// TIA Portal project "64396156_S7-1200_DataLogging_PROJ_v2d0" (V14)

(* hardware
DEVICE "SIMATIC 1200-Station_1"  S71200.Device
   slot 0: "S7-1200 rack"  Rack  V1.0
   slot 1: "PLC_1"  CPU 1211C DC/DC/DC  6ES7 211-1AE40-0XB0  V4.2
*)

// ===== PLC "PLC_1"  CPU 1211C DC/DC/DC =====

VAR_GLOBAL   // PLC tag table "Standard-Variablentabelle"
   "System_Byte" AT %MB1 : Byte;
   "FirstScan" AT %M1.0 : Bool;
   "DiagStatusUpdate" AT %M1.1 : Bool;
   "AlwaysTRUE" AT %M1.2 : Bool;
   "AlwaysFALSE" AT %M1.3 : Bool;
   "Clock_Byte" AT %MB0 : Byte;
   "Clock_10Hz" AT %M0.0 : Bool;
   "Clock_5Hz" AT %M0.1 : Bool;
   "Clock_2.5Hz" AT %M0.2 : Bool;
   "Clock_2Hz" AT %M0.3 : Bool;
   "Clock_1.25Hz" AT %M0.4 : Bool;
   "Clock_1Hz" AT %M0.5 : Bool;
   "Clock_0.625Hz" AT %M0.6 : Bool;
   "Clock_0.5Hz" AT %M0.7 : Bool;
END_VAR

TYPE "BLOCK"
VERSION : 0.1
   STRUCT
      REQ : Bool;
      DONE : Bool;
      BUSY : Bool;
      ERROR : Bool;
      STATUS : Word;
   END_STRUCT;
END_TYPE

TYPE "Type_SndParam"
VERSION : 0.1
   STRUCT
      interfaceId : Hw_Any;   // Hardware identifier
      conId : Conn_Ouc;   // Connection ID
      phoneNumber : String[22];   // Phone number
      smsText : String[160];   // Sms Text
   END_STRUCT;
END_TYPE

DATA_BLOCK "Tags"   // DB147
{ S7_Optimized_Access := 'TRUE' }
VERSION : 0.1
   VAR
      T : Struct
         Temperature : Real;
         Offset : Real := -22.0;
         Amplitude : Real := 6.0;
         Period : Real := 600.0;
      END_STRUCT;
   END_VAR
   VAR RETAIN
      DataLog : Struct
         Enable : Bool := true;
         Reset : Bool;
         DATA : Struct
            Temperature : Real;
         END_STRUCT;
         State : USInt;
         ErrorStatus : Word;
         NumberRecords : UDInt;
         CurrentName : String;
         WriteDone : Bool;
      END_STRUCT;
      TmailC : Struct
         Enable : Bool := false;
         Temperature_max : Real := -20.0;
         Reset : Bool;
         State : USInt;
         ErrorStatus : Word;
         ErrorCounter : UDInt;
         DoneCounter : UDInt;
      END_STRUCT;
   END_VAR
   VAR
      sms : Struct
         enable : Bool;
         sndSmsParam : "Type_SndParam";
         sndSmsOB1 : Bool;   // Bit, which activates Snd Sms block
         doneSndOB1 : Bool;   // Done. Signal for one progrmm cycle active
         busySndOB1 : Bool;   // Block is active
         errorSndOB1 : Bool;   // Error. Signal for one cycle active
         statusSndOB1 : DWord;   // Error Status for one Program cycle active
      END_STRUCT;
   END_VAR
BEGIN
   sms.sndSmsParam.smsText := 'The temperature is too high! Please check the system.';
   sms.sndSmsParam.phoneNumber := '+4915150006535';
   sms.sndSmsParam.conId := 1;
   sms.sndSmsParam.interfaceId := 270;
END_DATA_BLOCK

// folder: DataLog

DATA_BLOCK "DataLog_DB"   // DB143
{ S7_Optimized_Access := 'TRUE' }
VERSION : 0.1
// stored: InstanceOfName DataLog
"DataLog"
BEGIN
END_DATA_BLOCK

// folder: Simulation

DATA_BLOCK "T_simulation_DB"   // DB148
{ S7_Optimized_Access := 'TRUE' }
VERSION : 0.1
// stored: InstanceOfName T_simulation
"T_simulation"
BEGIN
END_DATA_BLOCK

// folder: TmailC

DATA_BLOCK "TmailC_DB"   // DB149
{ S7_Optimized_Access := 'TRUE' }
VERSION : 0.1
// stored: InstanceOfName TmailC
"TmailC"
BEGIN
END_DATA_BLOCK

// folder: (top level)

ORGANIZATION_BLOCK "Main"   // OB1, FBD, ProgramCycle
TITLE = "Main Program Sweep (Cycle)"
{ S7_Optimized_Access := 'TRUE' }
VERSION : 0.1
   VAR_INPUT
      Initial_Call : Bool;   // Initial call of this OB
      Remanence : Bool;   // =True, if remanent data are available
   END_VAR
BEGIN

REGION Network 1: Temperature simulation
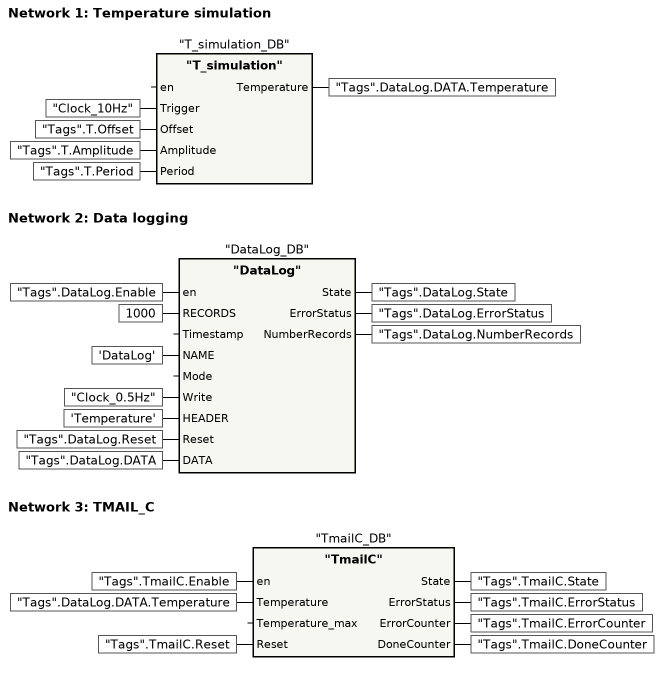
   "T_simulation_DB"(Trigger := "Clock_10Hz",   // "T_simulation"
                     Offset := "Tags".T.Offset,
                     Amplitude := "Tags".T.Amplitude,
                     Period := "Tags".T.Period,
                     Temperature => "Tags".DataLog.DATA.Temperature);
END_REGION

REGION Network 2: Data logging
   IF "Tags".DataLog.Enable THEN
       "DataLog_DB"(RECORDS := 1000,   // "DataLog"
                    "NAME" := 'DataLog',
                    Write := "Clock_0.5Hz",
                    HEADER := 'Temperature',
                    Reset := "Tags".DataLog.Reset,
                    DATA := "Tags".DataLog.DATA,
                    State => "Tags".DataLog.State,
                    ErrorStatus => "Tags".DataLog.ErrorStatus,
                    NumberRecords => "Tags".DataLog.NumberRecords);
   END_IF;
END_REGION

REGION Network 3: TMAIL_C
   IF "Tags".TmailC.Enable THEN
       "TmailC_DB"(Temperature := "Tags".DataLog.DATA.Temperature,   // "TmailC"
                   Reset := "Tags".TmailC.Reset,
                   State => "Tags".TmailC.State,
                   ErrorStatus => "Tags".TmailC.ErrorStatus,
                   ErrorCounter => "Tags".TmailC.ErrorCounter,
                   DoneCounter => "Tags".TmailC.DoneCounter);
   END_IF;
END_REGION
END_ORGANIZATION_BLOCK

// folder: DataLog

FUNCTION_BLOCK "DataLog"   // FB143, LAD
{ S7_Optimized_Access := 'TRUE' }
VERSION : 0.1
   VAR_INPUT
      RECORDS : UDInt;
      Timestamp : Bool := true;
      "NAME" : String;
      Mode : Bool;
      Write : Bool;
      HEADER : String;
      Reset : Bool;
   END_VAR
   VAR_OUTPUT
      State : USInt;
      ErrorStatus : Word;
      NumberRecords : UDInt;
   END_VAR
   VAR_IN_OUT
      DATA : Variant;
   END_VAR
   VAR RETAIN
      ID : UDInt;
      "Step" : USInt;
   END_VAR
   VAR
      CreateB : "BLOCK";
      OpenB : "BLOCK";
      WriteB : "BLOCK";
      write_edge : Bool;
   END_VAR
   VAR RETAIN
      NumberRecords_inout : UDInt;
   END_VAR
   VAR
      HEADER_inout : String;
      DataLogCreate_Instance : DataLogCreate;
      DataLogOpen_Instance : DataLogOpen;
      DataLogWrite_Instance : DataLogWrite;
      tmp_TIMESTAMP : UInt;
      tmp_MODE : UInt;
   END_VAR
   VAR_TEMP   // added for the SCL form of the ladder/FBD networks
      _w1 : Bool;
      _w2 : Bool;
      _w3 : Bool;
   END_VAR
BEGIN

REGION Network 1: Command 0: Create
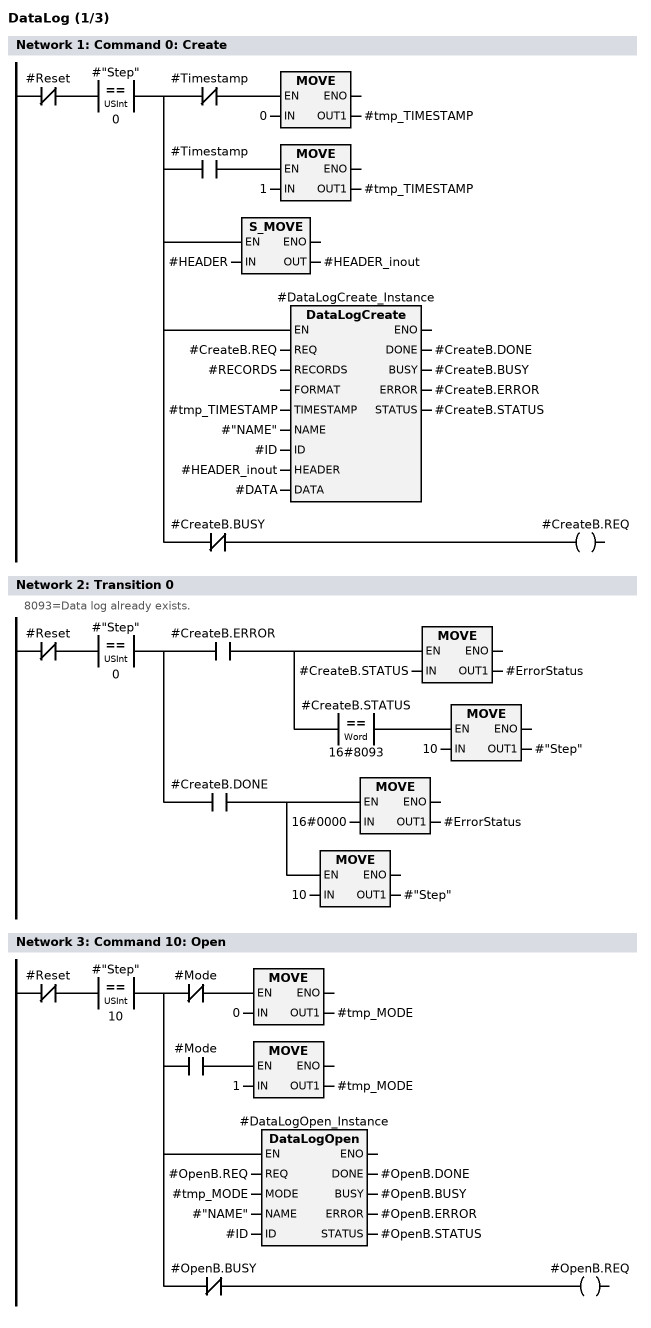
   #_w1 := NOT #Reset AND (#"Step" = 0);
   IF #_w1 AND NOT #Timestamp THEN #tmp_TIMESTAMP := 0; END_IF;
   IF #_w1 AND #Timestamp THEN #tmp_TIMESTAMP := 1; END_IF;
   IF #_w1 THEN
       #HEADER_inout := #HEADER;
       #DataLogCreate_Instance(REQ := #CreateB.REQ,   // DataLogCreate
                               RECORDS := #RECORDS,
                               TIMESTAMP := #tmp_TIMESTAMP,
                               "NAME" := #"NAME",
                               ID := #ID,
                               HEADER := #HEADER_inout,
                               DATA := #DATA,
                               DONE => #CreateB.DONE,
                               BUSY => #CreateB.BUSY,
                               ERROR => #CreateB.ERROR,
                               STATUS => #CreateB.STATUS);
   END_IF;
   #CreateB.REQ := #_w1 AND NOT #CreateB.BUSY;
END_REGION

REGION Network 2: Transition 0
   // 8093=Data log already exists.
   RUNG wire#powerrail
      I_Contact( #Reset )
      { S7_Templates := "SrcType := USInt" } EQ_Contact(in1 := #"Step", in2 := 0)
      wire#w1
      Contact( #CreateB.ERROR )
      wire#w2
      { S7_GenerateENO := "TRUE" } Move(in := #CreateB.STATUS, out1 => #ErrorStatus)
   END_RUNG
   RUNG wire#w2
      { S7_Templates := "SrcType := Word" } EQ_Contact(in1 := #CreateB.STATUS, in2 := 16#8093)
      { S7_GenerateENO := "TRUE" } Move(in := 10, out1 => #"Step")
   END_RUNG
   RUNG wire#w1
      Contact( #CreateB.DONE )
      wire#w3
      { S7_GenerateENO := "TRUE" } Move(in := 16#0000, out1 => #ErrorStatus)
   END_RUNG
   RUNG wire#w3
      { S7_GenerateENO := "TRUE" } Move(in := 10, out1 => #"Step")
   END_RUNG
   // the same network as SCL:
   #_w1 := NOT #Reset AND (#"Step" = 0);
   #_w2 := #_w1 AND #CreateB.ERROR;
   IF #_w2 THEN #ErrorStatus := #CreateB.STATUS; END_IF;
   IF #_w2 AND (#CreateB.STATUS = 16#8093) THEN #"Step" := 10; END_IF;
   IF #_w1 AND #CreateB.DONE THEN
       #ErrorStatus := 16#0000;
       #"Step" := 10;
   END_IF;
END_REGION

REGION Network 3: Command 10: Open
   #_w1 := NOT #Reset AND (#"Step" = 10);
   IF #_w1 AND NOT #Mode THEN #tmp_MODE := 0; END_IF;
   IF #_w1 AND #Mode THEN #tmp_MODE := 1; END_IF;
   IF #_w1 THEN
       #DataLogOpen_Instance(REQ := #OpenB.REQ,   // DataLogOpen
                             MODE := #tmp_MODE,
                             "NAME" := #"NAME",
                             ID := #ID,
                             DONE => #OpenB.DONE,
                             BUSY => #OpenB.BUSY,
                             ERROR => #OpenB.ERROR,
                             STATUS => #OpenB.STATUS);
   END_IF;
   #OpenB.REQ := #_w1 AND NOT #OpenB.BUSY;
END_REGION

REGION Network 4: Transition 10
   // 8092=Data log does not exist
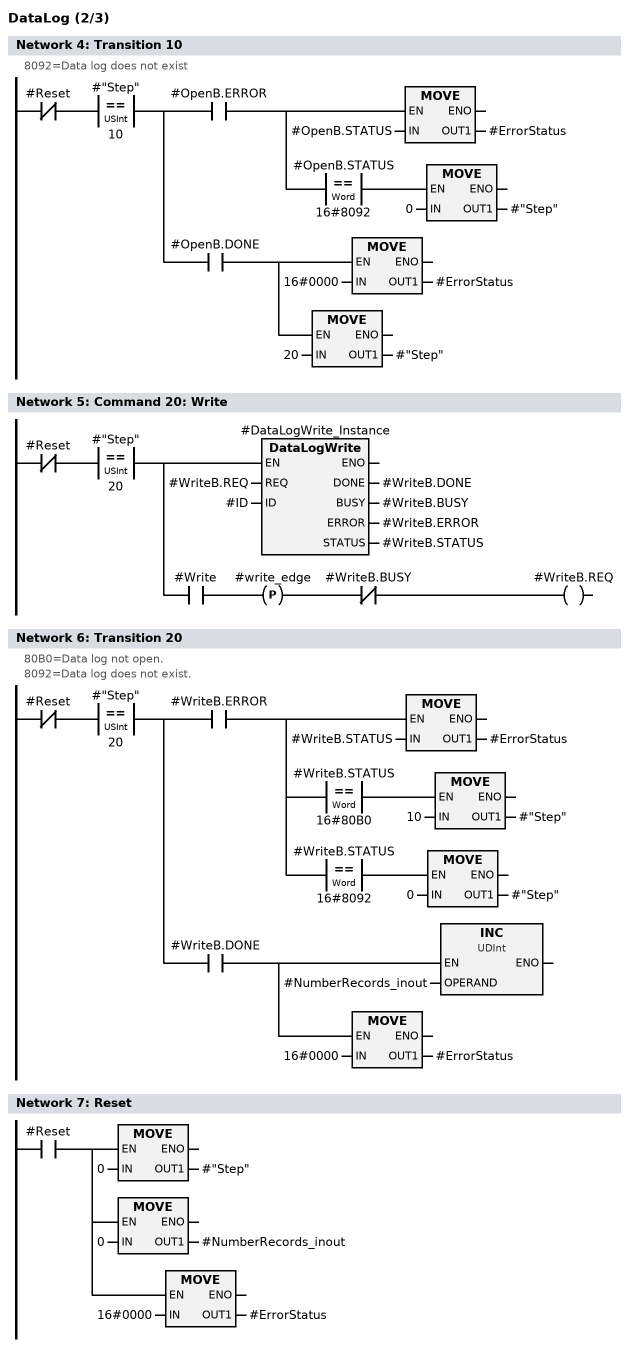
   RUNG wire#powerrail
      I_Contact( #Reset )
      { S7_Templates := "SrcType := USInt" } EQ_Contact(in1 := #"Step", in2 := 10)
      wire#w1
      Contact( #OpenB.ERROR )
      wire#w2
      { S7_GenerateENO := "TRUE" } Move(in := #OpenB.STATUS, out1 => #ErrorStatus)
   END_RUNG
   RUNG wire#w2
      { S7_Templates := "SrcType := Word" } EQ_Contact(in1 := #OpenB.STATUS, in2 := 16#8092)
      { S7_GenerateENO := "TRUE" } Move(in := 0, out1 => #"Step")
   END_RUNG
   RUNG wire#w1
      Contact( #OpenB.DONE )
      wire#w3
      { S7_GenerateENO := "TRUE" } Move(in := 16#0000, out1 => #ErrorStatus)
   END_RUNG
   RUNG wire#w3
      { S7_GenerateENO := "TRUE" } Move(in := 20, out1 => #"Step")
   END_RUNG
   // the same network as SCL:
   #_w1 := NOT #Reset AND (#"Step" = 10);
   #_w2 := #_w1 AND #OpenB.ERROR;
   IF #_w2 THEN #ErrorStatus := #OpenB.STATUS; END_IF;
   IF #_w2 AND (#OpenB.STATUS = 16#8092) THEN #"Step" := 0; END_IF;
   IF #_w1 AND #OpenB.DONE THEN
       #ErrorStatus := 16#0000;
       #"Step" := 20;
   END_IF;
END_REGION

REGION Network 5: Command 20: Write
   #_w1 := NOT #Reset AND (#"Step" = 20);
   IF #_w1 THEN
       #DataLogWrite_Instance(REQ := #WriteB.REQ,   // DataLogWrite
                              ID := #ID,
                              DONE => #WriteB.DONE,
                              BUSY => #WriteB.BUSY,
                              ERROR => #WriteB.ERROR,
                              STATUS => #WriteB.STATUS);
   END_IF;
   #_w2 := #_w1 AND #Write;
   #_w3 := #_w2 AND NOT #write_edge;   // rising edge
   #write_edge := #_w2;
   #WriteB.REQ := #_w3 AND NOT #WriteB.BUSY;
END_REGION

REGION Network 6: Transition 20
   // 80B0=Data log not open.
   // 8092=Data log does not exist.
   RUNG wire#powerrail
      I_Contact( #Reset )
      { S7_Templates := "SrcType := USInt" } EQ_Contact(in1 := #"Step", in2 := 20)
      wire#w1
      Contact( #WriteB.ERROR )
      wire#w2
      { S7_GenerateENO := "TRUE" } Move(in := #WriteB.STATUS, out1 => #ErrorStatus)
   END_RUNG
   RUNG wire#w2
      { S7_Templates := "SrcType := Word" } EQ_Contact(in1 := #WriteB.STATUS, in2 := 16#80B0)
      { S7_GenerateENO := "TRUE" } Move(in := 10, out1 => #"Step")
   END_RUNG
   RUNG wire#w2
      { S7_Templates := "SrcType := Word" } EQ_Contact(in1 := #WriteB.STATUS, in2 := 16#8092)
      { S7_GenerateENO := "TRUE" } Move(in := 0, out1 => #"Step")
   END_RUNG
   RUNG wire#w1
      Contact( #WriteB.DONE )
      wire#w3
      { S7_Templates := "DestType := UDInt"; S7_GenerateENO := "TRUE" } Inc( #NumberRecords_inout )
   END_RUNG
   RUNG wire#w3
      { S7_GenerateENO := "TRUE" } Move(in := 16#0000, out1 => #ErrorStatus)
   END_RUNG
   // the same network as SCL:
   #_w1 := NOT #Reset AND (#"Step" = 20);
   #_w2 := #_w1 AND #WriteB.ERROR;
   IF #_w2 THEN #ErrorStatus := #WriteB.STATUS; END_IF;
   IF #_w2 AND (#WriteB.STATUS = 16#80B0) THEN #"Step" := 10; END_IF;
   IF #_w2 AND (#WriteB.STATUS = 16#8092) THEN #"Step" := 0; END_IF;
   IF #_w1 AND #WriteB.DONE THEN
       #NumberRecords_inout := #NumberRecords_inout + 1;
       #ErrorStatus := 16#0000;
   END_IF;
END_REGION

REGION Network 7: Reset
   RUNG wire#powerrail
      Contact( #Reset )
      wire#w1
      { S7_GenerateENO := "TRUE" } Move(in := 0, out1 => #"Step")
   END_RUNG
   RUNG wire#w1
      { S7_GenerateENO := "TRUE" } Move(in := 0, out1 => #NumberRecords_inout)
   END_RUNG
   RUNG wire#w1
      { S7_GenerateENO := "TRUE" } Move(in := 16#0000, out1 => #ErrorStatus)
   END_RUNG
   // the same network as SCL:
   IF #Reset THEN
       #"Step" := 0;
       #NumberRecords_inout := 0;
       #ErrorStatus := 16#0000;
   END_IF;
END_REGION

REGION Network 8: output
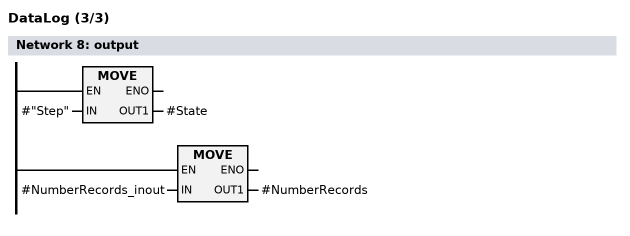
   RUNG wire#powerrail
      { S7_GenerateENO := "TRUE" } Move(in := #"Step", out1 => #State)
   END_RUNG
   RUNG wire#powerrail
      { S7_GenerateENO := "TRUE" } Move(in := #NumberRecords_inout, out1 => #NumberRecords)
   END_RUNG
   // the same network as SCL:
   #State := #"Step";
   #NumberRecords := #NumberRecords_inout;
END_REGION
END_FUNCTION_BLOCK

FUNCTION_BLOCK "DataLog_NewFile"   // FB145, LAD
{ S7_Optimized_Access := 'TRUE' }
VERSION : 0.1
   VAR_INPUT
      RECORDS : UDInt;
      Timestamp : Bool := true;
      "NAME" : String;
      Mode : Bool;
      Write : Bool;
      HEADER : String;
      NewFile_max : USInt := 30;
      Reset : Bool;
   END_VAR
   VAR_OUTPUT
      State : USInt;
      ErrorStatus : Word;
      NumberRecords : UDInt;
      CurrentName : String;
   END_VAR
   VAR_IN_OUT
      DATA : Variant;
   END_VAR
   VAR RETAIN
      Create_ID : UDInt;
      Open_ID : UDInt;
      NewFile_ID : UDInt;
      "Step" : USInt;
   END_VAR
   VAR
      CreateB : "BLOCK";
      OpenB : "BLOCK";
      WriteB : "BLOCK";
      CloseB : "BLOCK";
      NewFileB : "BLOCK";
      write_edge : Bool;
   END_VAR
   VAR RETAIN
      NewNumber : USInt := 1;
   END_VAR
   VAR
      Size : USInt;
      NewNumber_String : String;
   END_VAR
   VAR RETAIN
      NewFile_NAME : String;
      Open_NAME : String;
      NumberRecords_inout : UDInt;
   END_VAR
   VAR
      HEADER_inout : String;
      DataLogCreate_Instance : DataLogCreate;
      DataLogOpen_Instance : DataLogOpen;
      DataLogWrite_Instance : DataLogWrite;
      DataLogClose_Instance : DataLogClose;
      DataLogNewFile_Instance : DataLogNewFile;
      tmp_TIMESTAMP : USInt;
      tmp_MODE : UInt;
      tmp_SIZE : Real;
   END_VAR
   VAR_TEMP   // added for the SCL form of the ladder/FBD networks
      _w1 : Bool;
      _w2 : Bool;
      _w3 : Bool;
      _w4 : Bool;
   END_VAR
BEGIN

REGION Network 1: Command 0: Create
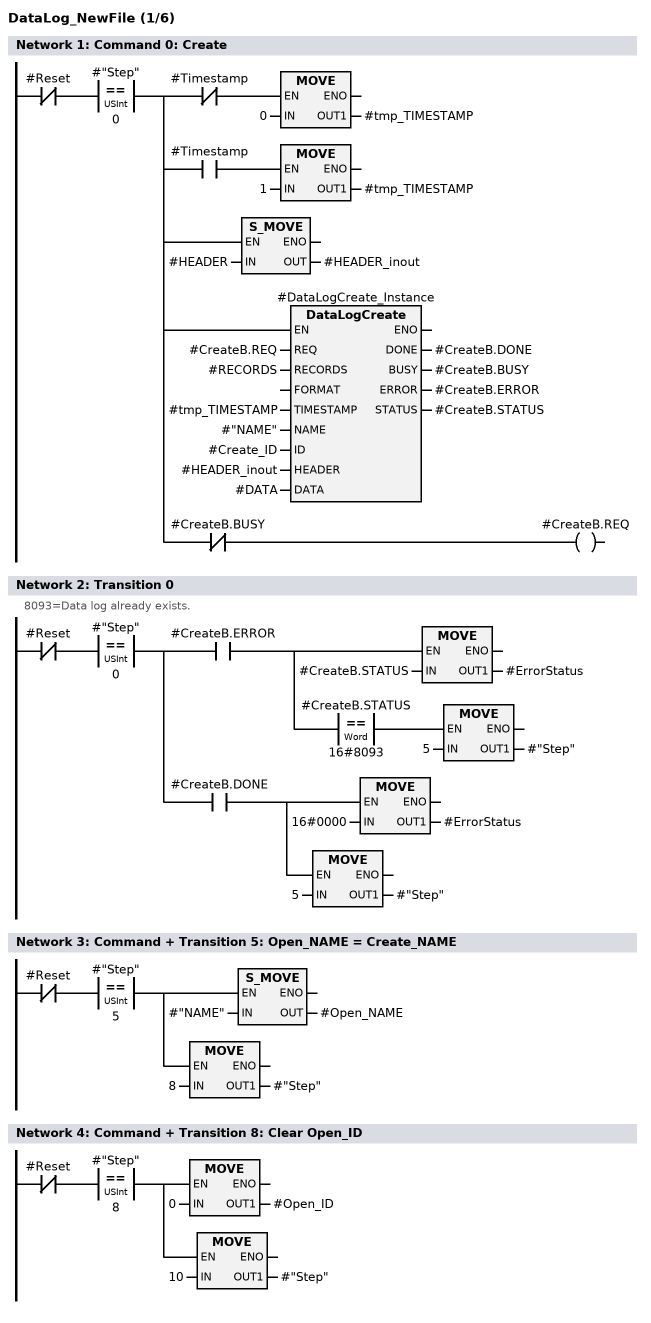
   #_w1 := NOT #Reset AND (#"Step" = 0);
   IF #_w1 AND NOT #Timestamp THEN #tmp_TIMESTAMP := 0; END_IF;
   IF #_w1 AND #Timestamp THEN #tmp_TIMESTAMP := 1; END_IF;
   IF #_w1 THEN
       #HEADER_inout := #HEADER;
       #DataLogCreate_Instance(REQ := #CreateB.REQ,   // DataLogCreate
                               RECORDS := #RECORDS,
                               TIMESTAMP := #tmp_TIMESTAMP,
                               "NAME" := #"NAME",
                               ID := #Create_ID,
                               HEADER := #HEADER_inout,
                               DATA := #DATA,
                               DONE => #CreateB.DONE,
                               BUSY => #CreateB.BUSY,
                               ERROR => #CreateB.ERROR,
                               STATUS => #CreateB.STATUS);
   END_IF;
   #CreateB.REQ := #_w1 AND NOT #CreateB.BUSY;
END_REGION

REGION Network 2: Transition 0
   // 8093=Data log already exists.
   RUNG wire#powerrail
      I_Contact( #Reset )
      { S7_Templates := "SrcType := USInt" } EQ_Contact(in1 := #"Step", in2 := 0)
      wire#w1
      Contact( #CreateB.ERROR )
      wire#w2
      { S7_GenerateENO := "TRUE" } Move(in := #CreateB.STATUS, out1 => #ErrorStatus)
   END_RUNG
   RUNG wire#w2
      { S7_Templates := "SrcType := Word" } EQ_Contact(in1 := #CreateB.STATUS, in2 := 16#8093)
      { S7_GenerateENO := "TRUE" } Move(in := 5, out1 => #"Step")
   END_RUNG
   RUNG wire#w1
      Contact( #CreateB.DONE )
      wire#w3
      { S7_GenerateENO := "TRUE" } Move(in := 16#0000, out1 => #ErrorStatus)
   END_RUNG
   RUNG wire#w3
      { S7_GenerateENO := "TRUE" } Move(in := 5, out1 => #"Step")
   END_RUNG
   // the same network as SCL:
   #_w1 := NOT #Reset AND (#"Step" = 0);
   #_w2 := #_w1 AND #CreateB.ERROR;
   IF #_w2 THEN #ErrorStatus := #CreateB.STATUS; END_IF;
   IF #_w2 AND (#CreateB.STATUS = 16#8093) THEN #"Step" := 5; END_IF;
   IF #_w1 AND #CreateB.DONE THEN
       #ErrorStatus := 16#0000;
       #"Step" := 5;
   END_IF;
END_REGION

REGION Network 3: Command + Transition 5: Open_NAME = Create_NAME
   RUNG wire#powerrail
      I_Contact( #Reset )
      { S7_Templates := "SrcType := USInt" } EQ_Contact(in1 := #"Step", in2 := 5)
      wire#w1
      { S7_GenerateENO := "TRUE" } S_Move(in := #"NAME", out => #Open_NAME)
   END_RUNG
   RUNG wire#w1
      { S7_GenerateENO := "TRUE" } Move(in := 8, out1 => #"Step")
   END_RUNG
   // the same network as SCL:
   IF NOT #Reset AND (#"Step" = 5) THEN
       #Open_NAME := #"NAME";
       #"Step" := 8;
   END_IF;
END_REGION

REGION Network 4: Command + Transition 8: Clear Open_ID
   RUNG wire#powerrail
      I_Contact( #Reset )
      { S7_Templates := "SrcType := USInt" } EQ_Contact(in1 := #"Step", in2 := 8)
      wire#w1
      { S7_GenerateENO := "TRUE" } Move(in := 0, out1 => #Open_ID)
   END_RUNG
   RUNG wire#w1
      { S7_GenerateENO := "TRUE" } Move(in := 10, out1 => #"Step")
   END_RUNG
   // the same network as SCL:
   IF NOT #Reset AND (#"Step" = 8) THEN
       #Open_ID := 0;
       #"Step" := 10;
   END_IF;
END_REGION

REGION Network 5: Command 10: Open
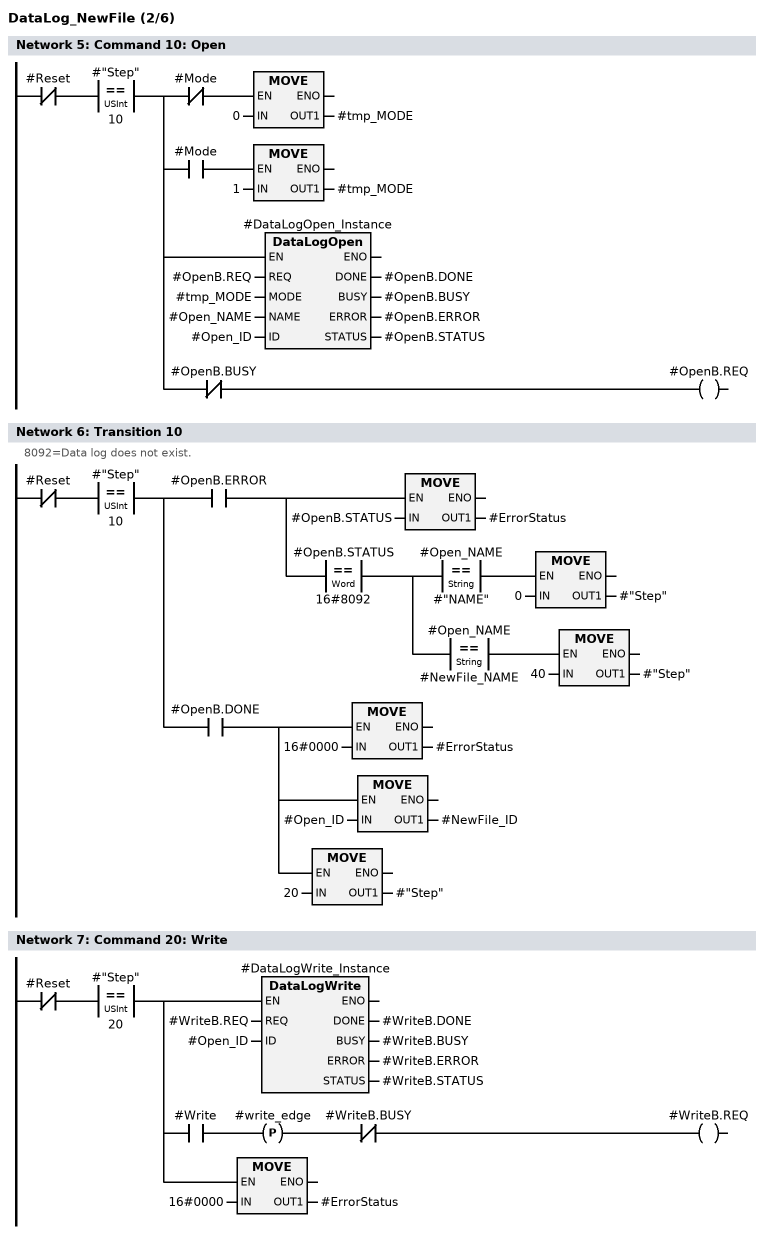
   #_w1 := NOT #Reset AND (#"Step" = 10);
   IF #_w1 AND NOT #Mode THEN #tmp_MODE := 0; END_IF;
   IF #_w1 AND #Mode THEN #tmp_MODE := 1; END_IF;
   IF #_w1 THEN
       #DataLogOpen_Instance(REQ := #OpenB.REQ,   // DataLogOpen
                             MODE := #tmp_MODE,
                             "NAME" := #Open_NAME,
                             ID := #Open_ID,
                             DONE => #OpenB.DONE,
                             BUSY => #OpenB.BUSY,
                             ERROR => #OpenB.ERROR,
                             STATUS => #OpenB.STATUS);
   END_IF;
   #OpenB.REQ := #_w1 AND NOT #OpenB.BUSY;
END_REGION

REGION Network 6: Transition 10
   // 8092=Data log does not exist.
   RUNG wire#powerrail
      I_Contact( #Reset )
      { S7_Templates := "SrcType := USInt" } EQ_Contact(in1 := #"Step", in2 := 10)
      wire#w1
      Contact( #OpenB.ERROR )
      wire#w2
      { S7_GenerateENO := "TRUE" } Move(in := #OpenB.STATUS, out1 => #ErrorStatus)
   END_RUNG
   RUNG wire#w2
      { S7_Templates := "SrcType := Word" } EQ_Contact(in1 := #OpenB.STATUS, in2 := 16#8092)
      wire#w3
      { S7_Templates := "SrcType := String" } EQ_Contact(in1 := #Open_NAME, in2 := #"NAME")
      { S7_GenerateENO := "TRUE" } Move(in := 0, out1 => #"Step")
   END_RUNG
   RUNG wire#w3
      { S7_Templates := "SrcType := String" } EQ_Contact(in1 := #Open_NAME, in2 := #NewFile_NAME)
      { S7_GenerateENO := "TRUE" } Move(in := 40, out1 => #"Step")
   END_RUNG
   RUNG wire#w1
      Contact( #OpenB.DONE )
      wire#w4
      { S7_GenerateENO := "TRUE" } Move(in := 16#0000, out1 => #ErrorStatus)
   END_RUNG
   RUNG wire#w4
      { S7_GenerateENO := "TRUE" } Move(in := #Open_ID, out1 => #NewFile_ID)
   END_RUNG
   RUNG wire#w4
      { S7_GenerateENO := "TRUE" } Move(in := 20, out1 => #"Step")
   END_RUNG
   // the same network as SCL:
   #_w1 := NOT #Reset AND (#"Step" = 10);
   #_w2 := #_w1 AND #OpenB.ERROR;
   IF #_w2 THEN #ErrorStatus := #OpenB.STATUS; END_IF;
   #_w3 := #_w2 AND (#OpenB.STATUS = 16#8092);
   IF #_w3 AND (#Open_NAME = #"NAME") THEN #"Step" := 0; END_IF;
   IF #_w3 AND (#Open_NAME = #NewFile_NAME) THEN #"Step" := 40; END_IF;
   IF #_w1 AND #OpenB.DONE THEN
       #ErrorStatus := 16#0000;
       #NewFile_ID := #Open_ID;
       #"Step" := 20;
   END_IF;
END_REGION

REGION Network 7: Command 20: Write
   #_w1 := NOT #Reset AND (#"Step" = 20);
   IF #_w1 THEN
       #DataLogWrite_Instance(REQ := #WriteB.REQ,   // DataLogWrite
                              ID := #Open_ID,
                              DONE => #WriteB.DONE,
                              BUSY => #WriteB.BUSY,
                              ERROR => #WriteB.ERROR,
                              STATUS => #WriteB.STATUS);
   END_IF;
   #_w2 := #_w1 AND #Write;
   #_w3 := #_w2 AND NOT #write_edge;   // rising edge
   #write_edge := #_w2;
   #WriteB.REQ := #_w3 AND NOT #WriteB.BUSY;
   IF #_w1 THEN #ErrorStatus := 16#0000; END_IF;
END_REGION

REGION Network 8: Transition 20
   // 80B0=Data log not open.
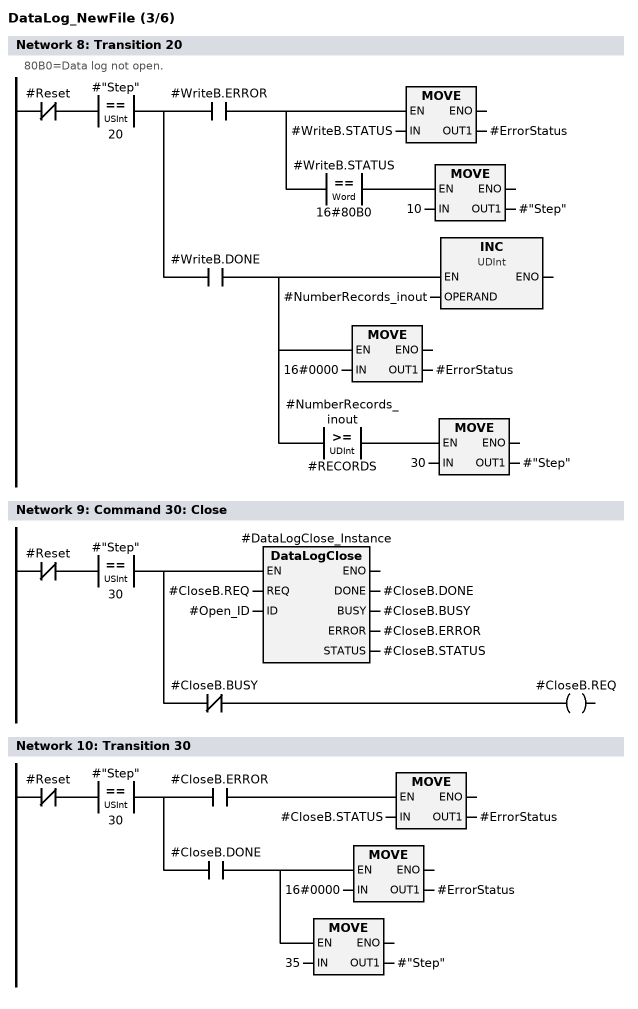
   RUNG wire#powerrail
      I_Contact( #Reset )
      { S7_Templates := "SrcType := USInt" } EQ_Contact(in1 := #"Step", in2 := 20)
      wire#w1
      Contact( #WriteB.ERROR )
      wire#w2
      { S7_GenerateENO := "TRUE" } Move(in := #WriteB.STATUS, out1 => #ErrorStatus)
   END_RUNG
   RUNG wire#w2
      { S7_Templates := "SrcType := Word" } EQ_Contact(in1 := #WriteB.STATUS, in2 := 16#80B0)
      { S7_GenerateENO := "TRUE" } Move(in := 10, out1 => #"Step")
   END_RUNG
   RUNG wire#w1
      Contact( #WriteB.DONE )
      wire#w3
      { S7_Templates := "DestType := UDInt"; S7_GenerateENO := "TRUE" } Inc( #NumberRecords_inout )
   END_RUNG
   RUNG wire#w3
      { S7_GenerateENO := "TRUE" } Move(in := 16#0000, out1 => #ErrorStatus)
   END_RUNG
   RUNG wire#w3
      { S7_Templates := "SrcType := UDInt" } GE_Contact(in1 := #NumberRecords_inout, in2 := #RECORDS)
      { S7_GenerateENO := "TRUE" } Move(in := 30, out1 => #"Step")
   END_RUNG
   // the same network as SCL:
   #_w1 := NOT #Reset AND (#"Step" = 20);
   #_w2 := #_w1 AND #WriteB.ERROR;
   IF #_w2 THEN #ErrorStatus := #WriteB.STATUS; END_IF;
   IF #_w2 AND (#WriteB.STATUS = 16#80B0) THEN #"Step" := 10; END_IF;
   #_w3 := #_w1 AND #WriteB.DONE;
   IF #_w3 THEN
       #NumberRecords_inout := #NumberRecords_inout + 1;
       #ErrorStatus := 16#0000;
   END_IF;
   IF #_w3 AND (#NumberRecords_inout >= #RECORDS) THEN #"Step" := 30; END_IF;
END_REGION

REGION Network 9: Command 30: Close
   #_w1 := NOT #Reset AND (#"Step" = 30);
   IF #_w1 THEN
       #DataLogClose_Instance(REQ := #CloseB.REQ,   // DataLogClose
                              ID := #Open_ID,
                              DONE => #CloseB.DONE,
                              BUSY => #CloseB.BUSY,
                              ERROR => #CloseB.ERROR,
                              STATUS => #CloseB.STATUS);
   END_IF;
   #CloseB.REQ := #_w1 AND NOT #CloseB.BUSY;
END_REGION

REGION Network 10: Transition 30
   RUNG wire#powerrail
      I_Contact( #Reset )
      { S7_Templates := "SrcType := USInt" } EQ_Contact(in1 := #"Step", in2 := 30)
      wire#w1
      Contact( #CloseB.ERROR )
      { S7_GenerateENO := "TRUE" } Move(in := #CloseB.STATUS, out1 => #ErrorStatus)
   END_RUNG
   RUNG wire#w1
      Contact( #CloseB.DONE )
      wire#w2
      { S7_GenerateENO := "TRUE" } Move(in := 16#0000, out1 => #ErrorStatus)
   END_RUNG
   RUNG wire#w2
      { S7_GenerateENO := "TRUE" } Move(in := 35, out1 => #"Step")
   END_RUNG
   // the same network as SCL:
   #_w1 := NOT #Reset AND (#"Step" = 30);
   IF #_w1 AND #CloseB.ERROR THEN #ErrorStatus := #CloseB.STATUS; END_IF;
   IF #_w1 AND #CloseB.DONE THEN
       #ErrorStatus := 16#0000;
       #"Step" := 35;
   END_IF;
END_REGION

REGION Network 11: Command + Transition 35: Create new file NAME
   // .
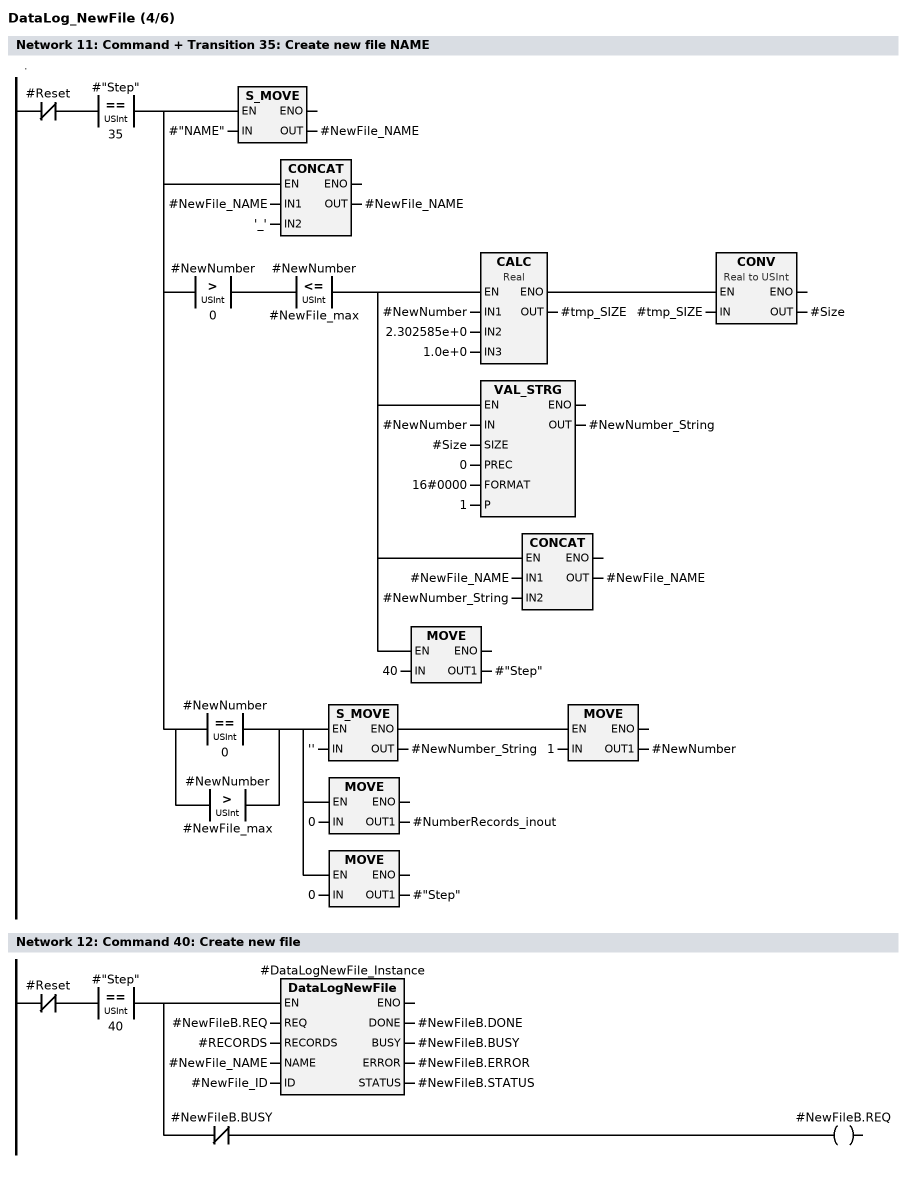
   // ENO of a box is taken as its EN; it also drops when the box reports an error
   #_w1 := NOT #Reset AND (#"Step" = 35);
   IF #_w1 THEN
       S_MOVE(in := #"NAME", out => #NewFile_NAME);
       #NewFile_NAME := CONCAT(IN1 := #NewFile_NAME, IN2 := '_');
   END_IF;
   #_w2 := #_w1 AND (#NewNumber > 0) AND (#NewNumber <= #NewFile_max);
   #_w3 := #_w1 AND (#NewNumber > 0) AND (#NewNumber <= #NewFile_max);
   IF #_w3 THEN
       CALC(in1 := #NewNumber, in2 := 2.302585e+0, in3 := 1.0e+0, out => #tmp_SIZE);
       #Size := REAL_TO_USINT(#tmp_SIZE);
   END_IF;
   IF #_w2 THEN
       VAL_STRG(IN := #NewNumber, SIZE := #Size, PREC := 0, FORMAT := 16#0000, P := 1, OUT => #NewNumber_String);
       #NewFile_NAME := CONCAT(IN1 := #NewFile_NAME, IN2 := #NewNumber_String);
       #"Step" := 40;
   END_IF;
   IF #_w1 AND ((#NewNumber = 0) OR (#NewNumber > #NewFile_max)) THEN
       S_MOVE(in := '', out => #NewNumber_String);
   END_IF;
   #_w4 := #_w1 AND ((#NewNumber = 0) OR (#NewNumber > #NewFile_max));
   IF #_w4 THEN
       #NewNumber := 1;
       #NumberRecords_inout := 0;
       #"Step" := 0;
   END_IF;
END_REGION

REGION Network 12: Command 40: Create new file
   #_w1 := NOT #Reset AND (#"Step" = 40);
   IF #_w1 THEN
       #DataLogNewFile_Instance(REQ := #NewFileB.REQ,   // DataLogNewFile
                               RECORDS := #RECORDS,
                               "NAME" := #NewFile_NAME,
                               ID := #NewFile_ID,
                               DONE => #NewFileB.DONE,
                               BUSY => #NewFileB.BUSY,
                               ERROR => #NewFileB.ERROR,
                               STATUS => #NewFileB.STATUS);
   END_IF;
   #NewFileB.REQ := #_w1 AND NOT #NewFileB.BUSY;
END_REGION

REGION Network 13: Transition 40
   // 8093=Data log already exists.
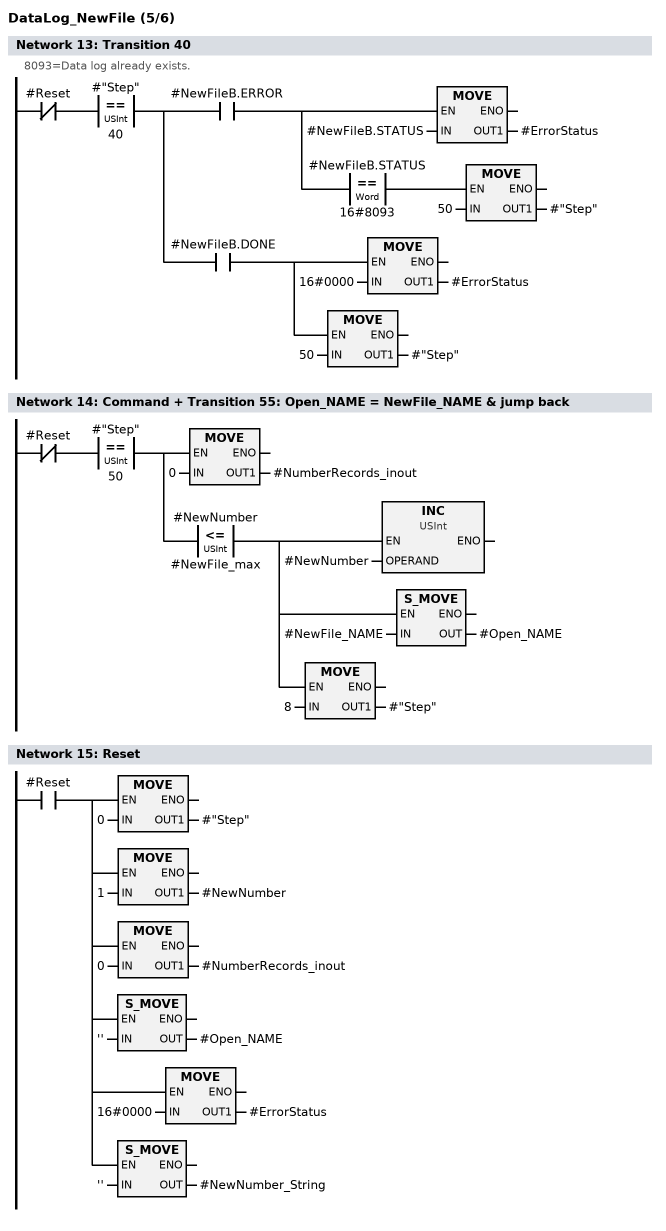
   RUNG wire#powerrail
      I_Contact( #Reset )
      { S7_Templates := "SrcType := USInt" } EQ_Contact(in1 := #"Step", in2 := 40)
      wire#w1
      Contact( #NewFileB.ERROR )
      wire#w2
      { S7_GenerateENO := "TRUE" } Move(in := #NewFileB.STATUS, out1 => #ErrorStatus)
   END_RUNG
   RUNG wire#w2
      { S7_Templates := "SrcType := Word" } EQ_Contact(in1 := #NewFileB.STATUS, in2 := 16#8093)
      { S7_GenerateENO := "TRUE" } Move(in := 50, out1 => #"Step")
   END_RUNG
   RUNG wire#w1
      Contact( #NewFileB.DONE )
      wire#w3
      { S7_GenerateENO := "TRUE" } Move(in := 16#0000, out1 => #ErrorStatus)
   END_RUNG
   RUNG wire#w3
      { S7_GenerateENO := "TRUE" } Move(in := 50, out1 => #"Step")
   END_RUNG
   // the same network as SCL:
   #_w1 := NOT #Reset AND (#"Step" = 40);
   #_w2 := #_w1 AND #NewFileB.ERROR;
   IF #_w2 THEN #ErrorStatus := #NewFileB.STATUS; END_IF;
   IF #_w2 AND (#NewFileB.STATUS = 16#8093) THEN #"Step" := 50; END_IF;
   IF #_w1 AND #NewFileB.DONE THEN
       #ErrorStatus := 16#0000;
       #"Step" := 50;
   END_IF;
END_REGION

REGION Network 14: Command + Transition 55: Open_NAME = NewFile_NAME & jump back
   RUNG wire#powerrail
      I_Contact( #Reset )
      { S7_Templates := "SrcType := USInt" } EQ_Contact(in1 := #"Step", in2 := 50)
      wire#w1
      { S7_GenerateENO := "TRUE" } Move(in := 0, out1 => #NumberRecords_inout)
   END_RUNG
   RUNG wire#w1
      { S7_Templates := "SrcType := USInt" } LE_Contact(in1 := #NewNumber, in2 := #NewFile_max)
      wire#w2
      { S7_Templates := "DestType := USInt"; S7_GenerateENO := "TRUE" } Inc( #NewNumber )
   END_RUNG
   RUNG wire#w2
      { S7_GenerateENO := "TRUE" } S_Move(in := #NewFile_NAME, out => #Open_NAME)
   END_RUNG
   RUNG wire#w2
      { S7_GenerateENO := "TRUE" } Move(in := 8, out1 => #"Step")
   END_RUNG
   // the same network as SCL:
   #_w1 := NOT #Reset AND (#"Step" = 50);
   IF #_w1 THEN #NumberRecords_inout := 0; END_IF;
   #_w2 := #_w1 AND (#NewNumber <= #NewFile_max);
   IF #_w2 THEN
       #NewNumber := #NewNumber + 1;
       #Open_NAME := #NewFile_NAME;
       #"Step" := 8;
   END_IF;
END_REGION

REGION Network 15: Reset
   RUNG wire#powerrail
      Contact( #Reset )
      wire#w1
      { S7_GenerateENO := "TRUE" } Move(in := 0, out1 => #"Step")
   END_RUNG
   RUNG wire#w1
      { S7_GenerateENO := "TRUE" } Move(in := 1, out1 => #NewNumber)
   END_RUNG
   RUNG wire#w1
      { S7_GenerateENO := "TRUE" } Move(in := 0, out1 => #NumberRecords_inout)
   END_RUNG
   RUNG wire#w1
      { S7_GenerateENO := "TRUE" } S_Move(in := '', out => #Open_NAME)
   END_RUNG
   RUNG wire#w1
      { S7_GenerateENO := "TRUE" } Move(in := 16#0000, out1 => #ErrorStatus)
   END_RUNG
   RUNG wire#w1
      { S7_GenerateENO := "TRUE" } S_Move(in := '', out => #NewNumber_String)
   END_RUNG
   // the same network as SCL:
   IF #Reset THEN
       #"Step" := 0;
       #NewNumber := 1;
       #NumberRecords_inout := 0;
       #Open_NAME := '';
       #ErrorStatus := 16#0000;
       #NewNumber_String := '';
   END_IF;
END_REGION

REGION Network 16: output
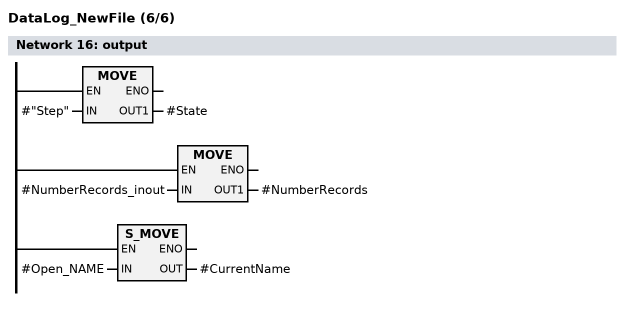
   RUNG wire#powerrail
      { S7_GenerateENO := "TRUE" } Move(in := #"Step", out1 => #State)
   END_RUNG
   RUNG wire#powerrail
      { S7_GenerateENO := "TRUE" } Move(in := #NumberRecords_inout, out1 => #NumberRecords)
   END_RUNG
   RUNG wire#powerrail
      { S7_GenerateENO := "TRUE" } S_Move(in := #Open_NAME, out => #CurrentName)
   END_RUNG
   // the same network as SCL:
   #State := #"Step";
   #NumberRecords := #NumberRecords_inout;
   #CurrentName := #Open_NAME;
END_REGION
END_FUNCTION_BLOCK

// folder: Simulation

FUNCTION_BLOCK "T_simulation"   // FB148, LAD
{ S7_Optimized_Access := 'TRUE' }
VERSION : 0.1
   VAR_INPUT
      Trigger : Bool;
      Offset : Real := -22.0;
      Amplitude : Real := 6.0;
      Period : Real := 600.0;
   END_VAR
   VAR_OUTPUT
      Temperature : Real;
   END_VAR
   VAR RETAIN
      "time" : Real := 0.0;
   END_VAR
   VAR
      Pi : Real := 3.141593;
      trigger_edge : Bool;
      "2_Pi" : Real;
   END_VAR
   VAR_TEMP   // added for the SCL form of the ladder/FBD networks
      _w1 : Bool;
   END_VAR
BEGIN

REGION Network 1
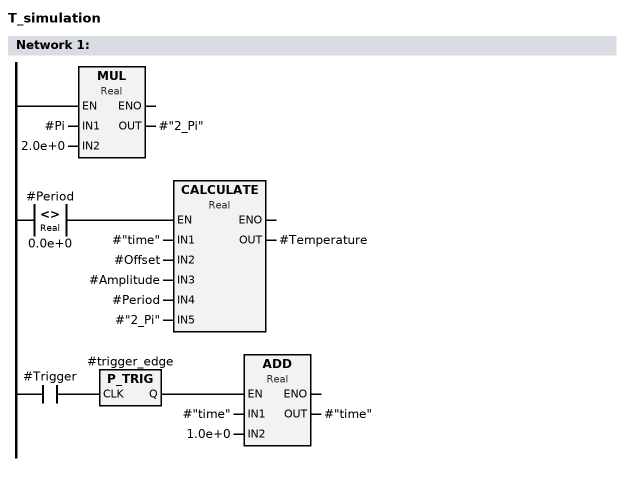
   RUNG wire#powerrail
      { S7_Templates := "SrcType := Real"; S7_GenerateENO := "TRUE" } Mul(in1 := #Pi, in2 := 2.0e+0, out => #"2_Pi")
   END_RUNG
   RUNG wire#powerrail
      { S7_Templates := "SrcType := Real" } NE_Contact(in1 := #Period, in2 := 0.0e+0)
      { S7_Templates := "SrcType := Real"; S7_GenerateENO := "TRUE"; S7_Expression := "IN2+IN3*Sin(IN1/IN4*IN5)" } Calculate(in1 := #"time", in2 := #Offset, in3 := #Amplitude, in4 := #Period, in5 := #"2_Pi", out => #Temperature)
   END_RUNG
   RUNG wire#powerrail
      Contact( #Trigger )
      P_Trig( #trigger_edge )
      { S7_Templates := "SrcType := Real"; S7_GenerateENO := "TRUE" } Add(in1 := #"time", in2 := 1.0e+0, out => #"time")
   END_RUNG
   // the same network as SCL:
   #"2_Pi" := #Pi * 2.0e+0;
   IF #Period <> 0.0e+0 THEN #Temperature := #Offset+#Amplitude*Sin(#"time"/#Period*#"2_Pi"); END_IF;
   #_w1 := #Trigger AND NOT #trigger_edge;   // rising edge
   #trigger_edge := #Trigger;
   IF #_w1 THEN #"time" := #"time" + 1.0e+0; END_IF;
END_REGION
END_FUNCTION_BLOCK

// folder: TmailC

FUNCTION_BLOCK "TmailC"   // FB149, FBD
{ S7_Optimized_Access := 'TRUE' }
VERSION : 0.1
   VAR_INPUT
      Temperature : Real;
      Temperature_max : Real := -20.0;
      Reset : Bool;
   END_VAR
   VAR_OUTPUT
      State : USInt;
      ErrorStatus : Word;
      ErrorCounter : UDInt;
      DoneCounter : UDInt;
   END_VAR
   VAR RETAIN
      "step" : USInt;
      ErrorCnt : UDInt;
      DoneCnt : UDInt;
      IEC_Timer_Instance : IEC_TIMER;
   END_VAR
   VAR
      DataLog_NewFile_Instance : "DataLog_NewFile";
   END_VAR
   VAR RETAIN
      TMAIL_C : "BLOCK";
      DataLog : Struct
         State : USInt;
         ErrorStatus : Word;
         NumberRecords : UDInt;
         CurrentName : String;
         DATA : Struct
            ERROR_STATUS : Word;
         END_STRUCT;
      END_STRUCT;
   END_VAR
   VAR
      TMAIL_C_Instance : TMAIL_C;
      tmailcMailAddrParam : TMail_V4;
   END_VAR
   VAR_TEMP   // added for the SCL form of the ladder/FBD networks
      _w1 : Bool;
   END_VAR
   // tmailcMailAddrParam.ID := 1;
   // tmailcMailAddrParam.MailServerAddress.ADDR[1] := 17;
   // tmailcMailAddrParam.MailServerAddress.ADDR[2] := 6;
   // tmailcMailAddrParam.MailServerAddress.ADDR[4] := 50;
   // tmailcMailAddrParam.WatchDogTime := T#1m;
   // tmailcMailAddrParam.UserName := 'gateway_account';
   // tmailcMailAddrParam.PassWord := 'password';
   // tmailcMailAddrParam.From.LocalPartPlusAtSign := 'gateway_account@';
   // tmailcMailAddrParam.From.FullQualifiedDomainName := 'gateway_server.com';
   // tmailcMailAddrParam.MailServerAddress.ADDR[3] := 1;
   // tmailcMailAddrParam.InterfaceId := 64;
   // tmailcMailAddrParam.ActiveEstablished := true;
BEGIN

REGION Network 1: TMAIL_C
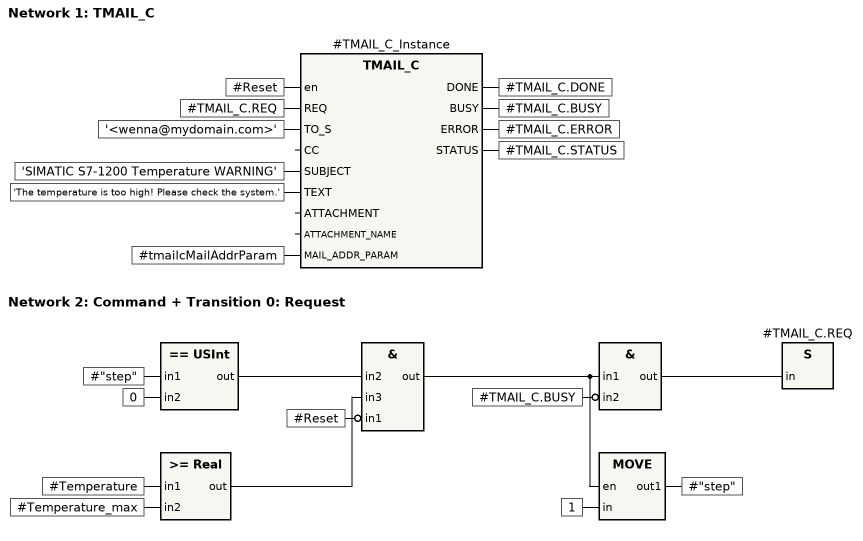
   IF #Reset THEN
       #TMAIL_C_Instance(REQ := #TMAIL_C.REQ,   // TMAIL_C
                         TO_S := '<wenna@mydomain.com>',
                         SUBJECT := 'SIMATIC S7-1200 Temperature WARNING',
                         TEXT := 'The temperature is too high! Please check the system.',
                         MAIL_ADDR_PARAM := #tmailcMailAddrParam,
                         DONE => #TMAIL_C.DONE,
                         BUSY => #TMAIL_C.BUSY,
                         ERROR => #TMAIL_C.ERROR,
                         STATUS => #TMAIL_C.STATUS);
   END_IF;
END_REGION

REGION Network 2: Command + Transition 0: Request
   #_w1 := (#"step" = 0) AND (#Temperature >= #Temperature_max) AND NOT #Reset;
   IF #_w1 AND NOT #TMAIL_C.BUSY THEN #TMAIL_C.REQ := TRUE; END_IF;
   IF #_w1 THEN #"step" := 1; END_IF;
END_REGION

REGION Network 3: Command + Transition 1: Switch Done / Error
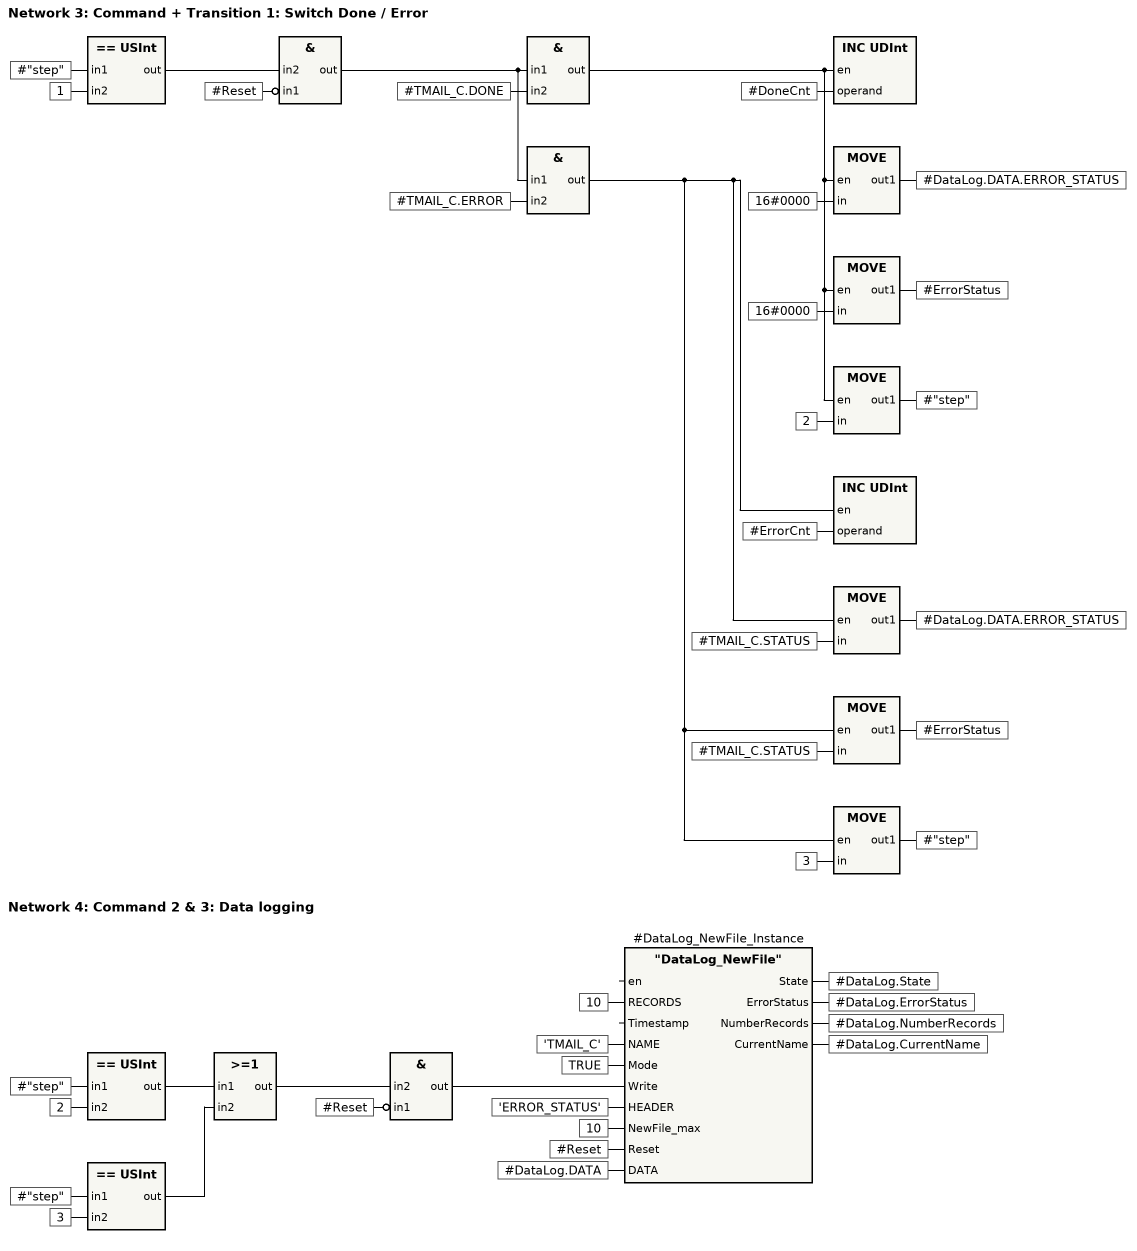
   #_w1 := (#"step" = 1) AND NOT #Reset;
   IF #_w1 AND #TMAIL_C.DONE THEN
       #DoneCnt := #DoneCnt + 1;
       #DataLog.DATA.ERROR_STATUS := 16#0000;
       #ErrorStatus := 16#0000;
       #"step" := 2;
   END_IF;
   IF #_w1 AND #TMAIL_C.ERROR THEN
       #ErrorCnt := #ErrorCnt + 1;
       #DataLog.DATA.ERROR_STATUS := #TMAIL_C.STATUS;
       #ErrorStatus := #TMAIL_C.STATUS;
       #"step" := 3;
   END_IF;
END_REGION

REGION Network 4: Command 2 & 3: Data logging
   #DataLog_NewFile_Instance(RECORDS := 10,   // "DataLog_NewFile"
                           "NAME" := 'TMAIL_C',
                           Mode := TRUE,
                           Write := ((#"step" = 2) OR (#"step" = 3)) AND NOT #Reset,
                           HEADER := 'ERROR_STATUS',
                           NewFile_max := 10,
                           Reset := #Reset,
                           DATA := #DataLog.DATA,
                           State => #DataLog.State,
                           ErrorStatus => #DataLog.ErrorStatus,
                           NumberRecords => #DataLog.NumberRecords,
                           CurrentName => #DataLog.CurrentName);
END_REGION

REGION Network 5: Transition 2 & 3: Write delay 100ms
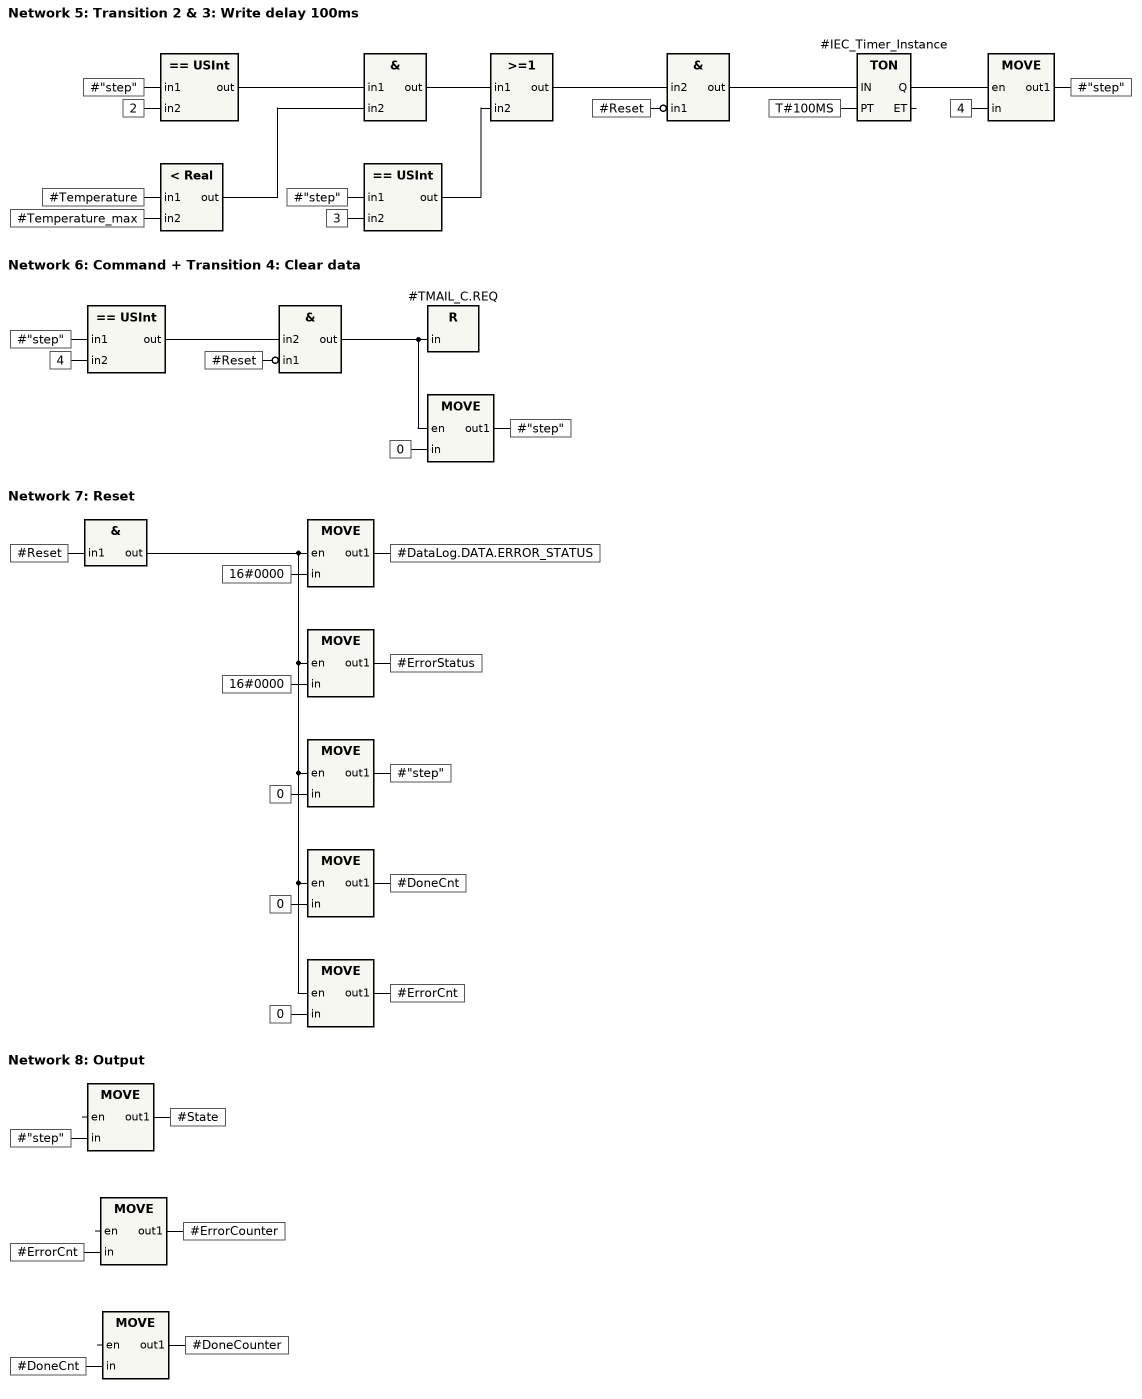
   #IEC_Timer_Instance.TON(IN := (((#"step" = 2) AND (#Temperature < #Temperature_max)) OR (#"step" = 3)) AND NOT #Reset,
                           PT := T#100MS);
   IF #IEC_Timer_Instance.Q THEN #"step" := 4; END_IF;
END_REGION

REGION Network 6: Command + Transition 4: Clear data
   IF (#"step" = 4) AND NOT #Reset THEN
       #TMAIL_C.REQ := FALSE;
       #"step" := 0;
   END_IF;
END_REGION

REGION Network 7: Reset
   IF #Reset THEN
       #DataLog.DATA.ERROR_STATUS := 16#0000;
       #ErrorStatus := 16#0000;
       #"step" := 0;
       #DoneCnt := 0;
       #ErrorCnt := 0;
   END_IF;
END_REGION

REGION Network 8: Output
   #State := #"step";
   #ErrorCounter := #ErrorCnt;
   #DoneCounter := #DoneCnt;
END_REGION
END_FUNCTION_BLOCK